% RSLogix 500 project PRJ_OUM_BAK018.RSS, saved by version 8.30.00.16 %
PROJECT "PRJ_OUM"    % processor: MicroLogix 1000 %

PROGRAM FILES
  LAD 2 "MAIN_PROG"  2 rungs
  LAD 3 "USER_FAULT"  1 rungs
  LAD 4 "HSC_INT"  1 rungs
  LAD 5 "STI_INT"  1 rungs
  LAD 6, 7, 8, 9, 10, 11, 12, 13, 14, 15, 16: only END

DATA FILES
  O0 OUTPUT  1 elements
  I1 INPUT  2 elements
  S2 STATUS  33 elements
  B3 BINARY  32 elements
  T4 TIMER  40 elements
  C5 COUNTER  32 elements
  R6 CONTROL  16 elements
  N7 INTEGER  105 elements

LADDER 2 "MAIN_PROG"
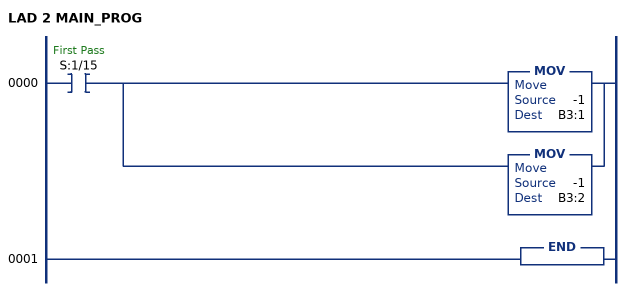
% Rung: 0 %
SOR XIC S:1/15 BST MOV -1 B3:1 NXB MOV -1 B3:2 BND EOR
%   S:1/15  "First Pass" %
% Rung: 1 %
SOR END EOR

OTHER DOCUMENTED ADDRESSES
  B3:0  B3
  B3:0/0  RES1_BAS
  B3:0/1  RES1_HAUT
  B3:0/2  RES2_BAS
  B3:0/3  RES2_HAUT
  B3:0/4  RES3_BAS
  B3:0/5  RES3_HAUT
  B3:0/6  RES4_BAS
  B3:0/7  RES4_HAUT
  FF  
  I:0.0/0  START
  O:0.0/0  POMP1_ON
  O:0.0/1  POMPE2_ON
  O:0.0/2  POMPE3_ON
  O:0.0/3  POMPE4_ON
  POMP2_ON  

DATA TABLE (non-zero values as saved)
DATA B3
% B3:0 % 0X0055 0X0000 0X0000 0X0000 0X0000 0X0000 0X0000 0X0000 0X0000 0X0000
